Yaskawa INFORM job: R1_W26(-90,90)(KAMERA).JBI

/JOB
//NAME R1_W26(-90,90)(KAMERA)
///FOLDERNAME SCIANA-NOWY-R2-KM
//POS
///NPOS 80,80,0,7,0,0
///TOOL 0
///POSTYPE PULSE
///PULSE
C00000=33159,-75041,-99219,-10449,70503,87317
C00001=75114,-71151,-88698,16556,84883,-79199
C00002=80306,-57576,-65743,15324,77013,-78443
C00003=81645,-55184,-62182,14985,75835,-78119
C00004=81645,-55158,-61101,15026,75205,-78199
C00005=81645,-55165,-61328,15018,75336,-78182
C00006=82615,-56161,-61879,14739,74994,-77878
C00007=81645,-55182,-62067,14991,75768,-78127
C00008=93593,2339,-24262,11010,80035,-73562
C00009=93896,1699,-22403,10959,78549,-73593
C00010=93896,1602,-21734,10976,78097,-73634
C00011=93896,1628,-21918,10972,78222,-73622
C00012=94601,1031,-22423,10744,78130,-73391
C00013=93896,1753,-22746,10951,78783,-73571
C00014=99701,55993,28634,9180,74385,-71946
C00015=100041,56388,31107,9120,73043,-71929
C00016=100041,56409,32034,9146,72491,-71971
C00017=100041,56403,31831,9140,72612,-71962
C00018=100636,55837,31197,8935,72644,-71751
C00019=100041,56386,31001,9117,73109,-71925
C00020=99543,52732,23022,9162,76158,-71867
C00021=97259,36235,-13419,9707,90177,-71548
C00022=112921,-101075,-101540,-5267,70967,-84838
C00023=131689,-94313,-78921,-26934,65320,-78038
C00024=125720,-68748,-64794,-24283,67507,-80950
C00025=125720,-68595,-63993,-24352,67129,-80866
C00026=125720,-68634,-64196,-24335,67226,-80887
C00027=124863,-68721,-64240,-24054,66961,-81168
C00028=125720,-68859,-65415,-24231,67808,-81013
C00029=125720,-69147,-67176,-24085,68663,-81201
C00030=124059,-7865,-28198,-22615,75116,-83143
C00031=124059,-8033,-26007,-22756,73788,-82883
C00032=124059,-8057,-25523,-22789,73503,-82829
C00033=124059,-8047,-25717,-22775,73619,-82852
C00034=123393,-8105,-25764,-22546,73438,-83063
C00035=124059,-7980,-26860,-22699,74300,-82986
C00036=124059,-7834,-28492,-22597,75300,-83178
C00037=123243,49055,25094,-22715,71613,-82758
C00038=123243,49133,27168,-22870,70468,-82530
C00039=123243,49200,28191,-22949,69918,-82418
C00040=123243,49185,27971,-22931,70034,-82441
C00041=122653,49127,27909,-22728,69882,-82636
C00042=123243,49111,26750,-22837,70695,-82574
C00043=123261,47208,21570,-22581,72747,-82975
C00044=127182,-103101,-86062,-25599,63792,-79509
C00045=127618,-116389,-73616,-42970,36666,-68730
C00046=127618,-115346,-72061,-43358,36354,-68513
C00047=125402,-115511,-72108,-42215,35270,-69391
C00048=125743,-96445,-78703,-25334,62336,-79769
C00049=125809,-92713,-74641,-25484,61829,-79621
C00050=125196,-75558,-67304,-24413,65559,-80740
C00051=124580,-57601,-58263,-23608,68741,-81673
C00052=124115,-41045,-48604,-23099,70972,-82311
C00053=123813,-29202,-40885,-22832,72126,-82656
C00054=123561,-15301,-30970,-22626,73021,-82929
C00055=123288,-2262,-20685,-22494,73291,-83084
C00056=123046,12399,-8053,-22436,73005,-83116
C00057=122891,24830,3475,-22463,72310,-83039
C00058=122733,39110,17699,-22574,70952,-82834
C00059=122600,54193,33794,-22815,68923,-82478
C00060=122491,72898,55194,-23336,65604,-81835
C00061=122584,71627,46958,-22691,69712,-82644
C00062=109861,33102,-26990,-2783,97255,-84296
C00063=100600,-79644,-90971,18148,89709,-63204
C00064=108129,-102348,-78221,22104,57738,-65711
C00065=110628,-102839,-78395,21205,56945,-64815
C00066=108411,-102755,-79295,21895,58084,-65517
C00067=110367,-78635,-73420,16519,77828,-61470
C00068=111567,-61213,-64952,16106,81188,-60595
C00069=112558,-45351,-55921,15823,83494,-59949
C00070=113363,-29331,-45716,15616,85224,-59450
C00071=113890,-16973,-36946,15493,86046,-59167
C00072=114365,-3321,-26319,15398,86417,-58960
C00073=114796,9401,-15539,15305,86245,-58833
C00074=115137,22724,-3341,15238,85542,-58805
C00075=115459,35185,8920,15184,84378,-58839
C00076=115787,51100,25673,15163,82258,-58985
C00077=116132,68210,45063,15202,79155,-59253
C00078=116103,68213,45043,15209,79173,-59261
C00079=116215,71808,25126,15033,92796,-57558
BC00000=206482,1287494,824008
BC00001=319465,1195750,1068222
BC00002=319465,1195750,1068222
BC00003=319465,1195750,1068222
BC00004=319465,1195750,1068222
BC00005=319465,1195750,1068222
BC00006=319465,1195750,1068222
BC00007=319465,1195750,1068222
BC00008=319465,1195750,1068222
BC00009=319465,1195750,1068222
BC00010=319465,1195750,1068222
BC00011=319465,1195750,1068222
BC00012=319465,1195750,1068222
BC00013=319465,1195750,1068222
BC00014=319465,1195750,1068222
BC00015=319465,1195750,1068222
BC00016=319465,1195750,1068222
BC00017=319465,1195750,1068222
BC00018=319465,1195750,1068222
BC00019=319465,1195750,1068222
BC00020=319465,1195750,1068222
BC00021=319465,1195750,1068222
BC00022=24752,1195750,1068222
BC00023=24752,1195750,1068222
BC00024=24752,1195750,1068222
BC00025=24752,1195750,1068222
BC00026=24752,1195750,1068222
BC00027=24752,1195750,1068222
BC00028=24752,1195750,1068222
BC00029=24752,1195750,1068222
BC00030=24752,1195750,1068222
BC00031=24752,1195750,1068222
BC00032=24752,1195750,1068222
BC00033=24752,1195750,1068222
BC00034=24752,1195750,1068222
BC00035=24752,1195750,1068222
BC00036=24752,1195750,1068222
BC00037=24752,1195750,1068222
BC00038=24752,1195750,1068222
BC00039=24752,1195750,1068222
BC00040=24752,1195750,1068222
BC00041=24752,1195750,1068222
BC00042=24752,1195750,1068222
BC00043=24752,1195750,1068222
BC00044=24752,1195750,1068222
BC00045=24752,1191142,1068222
BC00046=24752,1191142,1068222
BC00047=24752,1191142,1068222
BC00048=24752,1191142,1068222
BC00049=24752,1191142,1068222
BC00050=24752,1191142,1068222
BC00051=24752,1191142,1068222
BC00052=24752,1191142,1068222
BC00053=24752,1191142,1068222
BC00054=24752,1191142,1068222
BC00055=24752,1191142,1068222
BC00056=24752,1191142,1068222
BC00057=24752,1191142,1068222
BC00058=24752,1191142,1068222
BC00059=24752,1191142,1068222
BC00060=24752,1191142,1068222
BC00061=24752,1191142,1068222
BC00062=195212,1190663,1068222
BC00063=394654,1190102,1068223
BC00064=394654,1189027,1068223
BC00065=394654,1189027,1068223
BC00066=394654,1189027,1068223
BC00067=394654,1189027,1068223
BC00068=394654,1189029,1068221
BC00069=394654,1189029,1068221
BC00070=394654,1189029,1068221
BC00071=394654,1189029,1068221
BC00072=394654,1189029,1068219
BC00073=394654,1189029,1068219
BC00074=394654,1189029,1068219
BC00075=394654,1189029,1068219
BC00076=394654,1189029,1068219
BC00077=394654,1189029,1068219
BC00078=394654,1172585,1068219
BC00079=394654,1172585,1068219
///POSTYPE BASE
///RECTAN
///RCONF 0,0,0,0,0,0,0,0,0,0,0,0,0,0,0,0,0,0,0,0,0,0,0,0
P00006=0.222,-3.123,-1.508,0.0000,0.0000,0.0000
P00021=-0.225,-6.128,-0.405,0.0000,0.0000,0.0000
P00022=0.222,-3.123,-1.508,0.0000,0.0000,0.0000
P00023=0.143,-0.036,0.682,0.0000,0.0000,0.0000
P00024=0.145,-0.552,1.326,0.0000,0.0000,0.0000
P00025=-2.003,0.006,0.728,0.0000,0.0000,0.0000
P00026=0.562,-0.002,-0.337,0.0000,0.0000,0.0000
//INST
///DATE 2024/07/29 11:06
///ATTR SC,RW
///GROUP1 RB1,BS1
NOP
SFTOF
CALL JOB:ONLY_CUT_KM_NEW_SCIANA
SFTOF
MOVJ C00000 BC00000 VJ=100.00
MOVJ C00001 BC00001 VJ=100.00
MOVJ C00002 BC00002 VJ=100.00
'P1
MOVL C00003 BC00003 V=133.3
REFP 3 C00004 BC00004
CALL JOB:SEARCH-R1
SET P021 P006
SFTON P021
MOVL C00005 BC00005 V=66.7
REFP 3 C00006 BC00006
CALL JOB:SEARCH-R1
SET P021 P006
SFTON P021
MOVL C00007 BC00007 V=133.3
SFTOF
MOVL C00008 BC00008 V=1000.0
'P2
MOVL C00009 BC00009 V=133.3
REFP 3 C00010 BC00010
CALL JOB:SEARCH-R1
SET P022 P006
SFTON P022
MOVL C00011 BC00011 V=66.7
REFP 3 C00012 BC00012
CALL JOB:SEARCH-R1
SET P022 P006
SFTON P022
MOVL C00013 BC00013 V=133.3
SFTOF
MOVL C00014 BC00014 V=1000.0
'P3
MOVL C00015 BC00015 V=133.3
REFP 3 C00016 BC00016
CALL JOB:SEARCH-R1
SET P023 P006
SFTON P023
MOVL C00017 BC00017 V=83.3
REFP 3 C00018 BC00018
CALL JOB:SEARCH-R1
SET P023 P006
SFTON P023
MOVL C00019 BC00019 V=133.3
SFTOF
MOVL C00020 BC00020 V=1000.0
MOVJ C00021 BC00021 VJ=100.00
MOVJ C00022 BC00022 VJ=100.00
MOVJ C00023 BC00023 VJ=100.00
MOVL C00024 BC00024 V=133.3
'P1
REFP 3 C00025 BC00025
CALL JOB:SEARCH-R1
SET P024 P006
SFTON P024
MOVL C00026 BC00026 V=66.7
REFP 3 C00027 BC00027
CALL JOB:SEARCH-R1
SET P024 P006
SFTON P024
MOVL C00028 BC00028 V=133.3
SFTOF
MOVL C00029 BC00029 V=333.3
MOVL C00030 BC00030 V=1000.0
MOVL C00031 BC00031 V=133.3
'P2
REFP 3 C00032 BC00032
CALL JOB:SEARCH-R1
SET P025 P006
SFTON P025
MOVL C00033 BC00033 V=66.7
REFP 3 C00034 BC00034
CALL JOB:SEARCH-R1
SET P025 P006
SFTON P025
MOVL C00035 BC00035 V=133.3
SFTOF
MOVL C00036 BC00036 V=333.3
MOVL C00037 BC00037 V=333.3
MOVL C00038 BC00038 V=133.3
'P3
REFP 3 C00039 BC00039
CALL JOB:SEARCH-R1
SET P026 P006
SFTON P026
MOVL C00040 BC00040 V=66.7
REFP 3 C00041 BC00041
CALL JOB:SEARCH-R1
SET P026 P006
SFTON P026
MOVL C00042 BC00042 V=133.3
SFTOF
MOVL C00043 BC00043 V=333.3
MOVL C00044 BC00044 V=1000.0
MACRO1 MJ#(0) ARGF9
SFTON P024
MOVJ C00045 BC00045 VJ=100.00
MOVJ C00046 BC00046 VJ=25.00
ARCON
MOVL C00047 BC00047 V=11.0
ARCOF
MOVJ C00048 BC00048 VJ=25.00
MOVJ C00049 BC00049 VJ=15.00
MACRO1 MJ#(0) ARGF9
ARCON
MOVL C00050 BC00050 V=13.3
ARCOF
MOVL C00051 BC00051 V=41.7
ARCON
MOVL C00052 BC00052 V=13.3
ARCOF
SFTOF
SFTON P025
MOVL C00053 BC00053 V=83.3
ARCON
MOVL C00054 BC00054 V=13.3
ARCOF
MOVL C00055 BC00055 V=83.3
ARCON
MOVL C00056 BC00056 V=13.3
ARCOF
SFTOF
SFTON P026
MOVL C00057 BC00057 V=83.3
ARCON
MOVL C00058 BC00058 V=13.3
ARCOF
MOVL C00059 BC00059 V=83.3
ARCON
MOVL C00060 BC00060 V=16.7
ARCOF
MOVL C00061 BC00061 V=166.7
MOVJ C00062 BC00062 VJ=100.00
MOVJ C00063 BC00063 VJ=100.00
SFTON P021
MOVJ C00064 BC00064 VJ=25.00
ARCON
MOVL C00065 BC00065 V=11.0
ARCOF
MOVL C00066 BC00066 V=83.3
MOVL C00067 BC00067 V=166.7
ARCON
MOVL C00068 BC00068 V=13.3
ARCOF
MOVL C00069 BC00069 V=83.3
ARCON
MOVL C00070 BC00070 V=13.3
ARCOF
SFTOF
SFTON P022
MOVL C00071 BC00071 V=83.3
ARCON
MOVL C00072 BC00072 V=13.3
ARCOF
MOVL C00073 BC00073 V=83.3
ARCON
MOVL C00074 BC00074 V=13.3
ARCOF
SFTOF
SFTON P023
MOVL C00075 BC00075 V=83.3
ARCON
MOVL C00076 BC00076 V=13.3
ARCOF
MOVL C00077 BC00077 V=83.3
ARCON
MOVL C00078 BC00078 V=16.7
ARCOF
SFTOF
MOVL C00079 BC00079 V=166.7
END
